ABB RobotStudio station: 4_28 - Copy_20220202-173113.rsstn

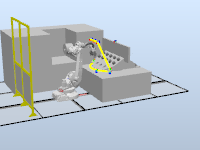
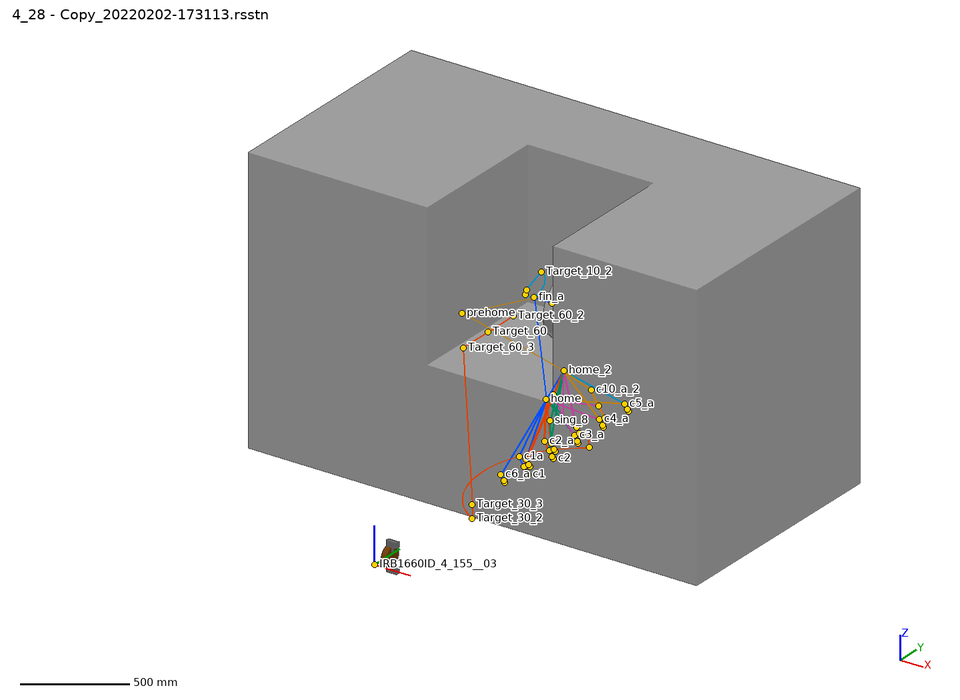
[picture v1: parts stored in the station drawn from their meshes, with robot base, taught points and paths (robot models come from the ABB library and are not in the file)]
Station Cambio_9_30 (saved by RobotStudio 21.4.9700.0)
Controller Controller3
  mechanical unit ROB_1: IRB1660ID_4_155__03, 6 joints, base frame (0, 0, 0) mm
Layout (positions relative to the parent item):
  - IRB1660ID_4_155__03 [mechanism, from Robots\IRB1660ID_4_155__03.rslib] at (0, 0, 0) mm; joint values [0.4367, 0.2271, -0.032, 0, 1.3757, 2.0075] (rad or m)
  - Pinza_1 [mechanism, from Efectores_finales - Copy\Pinza_1.rslib] at (900.75, 420.45, 1010) mm, rotated rx 180 ry 0 rz 90 deg; joint values [0, 0] (rad or m)
  - Conjunto_para_piezas_huecos [part] at (1981.81, -744.19, 0) mm, rotated rx 90 ry 0 rz 180 deg, size 1400 x 1300 x 1400 mm
  - Torno [part] at (-1172.42, 1966.27, 0) mm, rotated rx 0 ry 0 rz 180 deg, size 2500 x 1300 x 1500 mm
  - Fence_740 [graphiccomponentgroup, from Equipment\Fence_740.rslib] at (-1160.76, -802.49, 0) mm
    - Body 1 [part, from Equipment\Fence_740.rslib]
    - Body 2 [part, from Equipment\Fence_740.rslib]
  - Fence_2500 [graphiccomponentgroup, from Equipment\Fence_2500.rslib] at (1297.15, -826.85, 0) mm, rotated rx 0 ry 0 rz 90 deg
    - Body 1 [part, from Equipment\Fence_2500.rslib]
    - Body 2 [part, from Equipment\Fence_2500.rslib]
  - Fence_740_2 [graphiccomponentgroup, from Equipment\Fence_740.rslib] at (-1148.66, -57.63, 0) mm
    - Body 1 [part, from Equipment\Fence_740.rslib]
    - Body 2 [part, from Equipment\Fence_740.rslib]
  - c5 [part] at (1213.21, 355.81, 885.53) mm, rotated rx 0 ry -32 rz 0 deg, size 80 x 79.4 x 100 mm
  - c0 [part] at (367.03, 1016.09, 1000) mm, rotated rx -90 ry 0 rz 90 deg, size 80 x 79.4 x 100 mm
  - c8 [part] at (1084.59, -44.2, 808.36) mm, rotated rx 0 ry -32 rz 0 deg, size 80 x 79.4 x 100 mm
  - c4 [part] at (1213.21, 155.81, 885.53) mm, rotated rx 0 ry -32 rz 0 deg, size 80 x 79.4 x 100 mm
  - c7 [part] at (1084.59, -244.19, 808.36) mm, rotated rx 0 ry -32 rz 0 deg, size 80 x 79.4 x 100 mm
  - c6 [part] at (1084.59, -444.19, 808.36) mm, rotated rx 0 ry -32 rz 0 deg, size 80 x 79.4 x 100 mm
  - c9 [part] at (1084.59, 155.81, 808.36) mm, rotated rx 0 ry -32 rz 0 deg, size 80 x 79.4 x 100 mm
  - c10 [part] at (1084.59, 355.81, 808.36) mm, rotated rx 0 ry -32 rz 0 deg, size 80 x 79.4 x 100 mm
  - fin [part] at (377.58, 1016.27, 1000) mm, size 100 x 79.4 x 80 mm
  - c1 [part] at (1160.22, -444.2, 970.34) mm, rotated rx 90 ry 58 rz 0 deg, size 100 x 79.4 x 80 mm
  - Efector final 2 [part] at (70, 0, -80) mm, rotated rx 0 ry -90 rz -180 deg, size 100 x 99.5 x 30 mm
  - Pinza1_5 [part] at (130, 10, -10) mm, rotated rx 0 ry 0 rz 180 deg, size 60 x 20 x 60 mm
  - Pinza1_6 [part] at (130, -10, 150) mm, rotated rx 180 ry 0 rz 180 deg, size 60 x 20 x 60 mm
    - Pinza_2_1 [frame] at (30, 10, 80) mm, rotated rx 0 ry -90 rz 0 deg
  - Pinza_2 [mechanism, from Efectores_finales\PINZA2.rslib] at (900.75, 420.45, 1010) mm, rotated rx 180 ry 0 rz 90 deg; joint values [0, 0] (rad or m)
  - CollisionSensor [smart component, from Components\CollisionSensor.rslib]
      properties: Object1=Pinza_2; Object2=(none); NearMiss=0.0001; Part1=(none); Part2=(none); CollisionType=0
  - CollisionSensor_2 [smart component, from Components\CollisionSensor.rslib]
      properties: Object1=Pinza_2; Object2=c0_invisible; NearMiss=0.01; Part1=(none); Part2=(none); CollisionType=0
  - Attacher [smart component, from Components\Attacher.rslib]
      properties: Parent=Pinza_2; Flange=0; Child=(none); Mount=false; Offset=[0 0 0]; Orientation=[0 0 0]
  - Detacher [smart component, from Components\Detacher.rslib]
      properties: Child=(none); KeepPosition=true
  - CollisionSensor_3 [smart component, from Components\CollisionSensor.rslib]
      properties: Object1=Pinza_1; Object2=(none); NearMiss=0; Part1=(none); Part2=(none); CollisionType=0
  - Attacher_2 [smart component, from Components\Attacher.rslib]
      properties: Parent=Pinza_1; Flange=0; Child=(none); Mount=false; Offset=[0 0 0]; Orientation=[0 0 0]
  - Detacher_2 [smart component, from Components\Detacher.rslib]
      properties: Child=(none); KeepPosition=true
  - c2 [part] at (1207.14, -244.2, 895.25) mm, rotated rx 0 ry -32 rz 0 deg, size 80 x 79.4 x 100 mm
  - c0_invisible [part] at (277.58, 1016.27, 1000) mm, size 100 x 79.4 x 80 mm
  - CollisionSensor_4 [smart component, from Components\CollisionSensor.rslib]
      properties: Object1=Pinza_1; Object2=Conjunto_para_piezas_huecos; NearMiss=0.02; Part1=(none); Part2=(none); CollisionType=0
  - c3 [part] at (1213.21, -44.2, 885.53) mm, rotated rx 0 ry -32 rz 0 deg, size 80 x 79.4 x 100 mm
  - Hide [smart component, from Components\Hide.rslib]
      properties: Object=(none)
  - Show_2 [smart component, from Components\Show.rslib]
      properties: Object=Conjunto_para_piezas_huecos
  - visibilidad cilindros [smart component]
      signals: DI hide, DI show
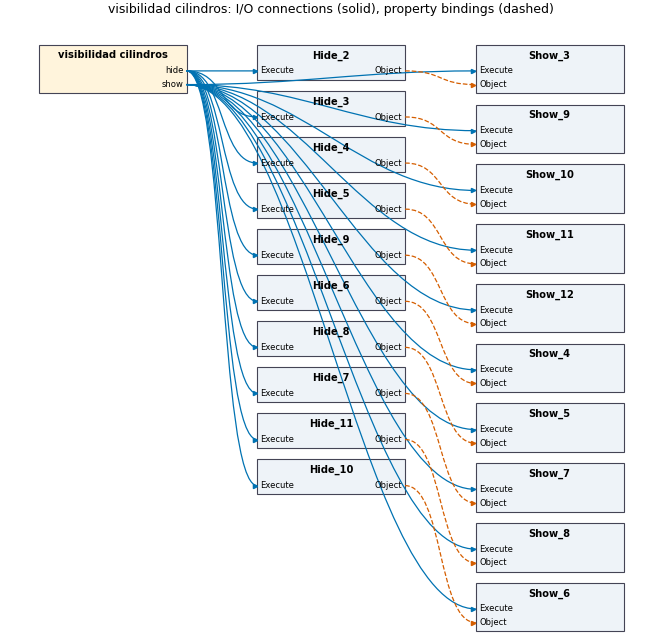
      connections:
        visibilidad cilindros.hide -> Hide_2.Execute
        visibilidad cilindros.hide -> Hide_3.Execute
        visibilidad cilindros.hide -> Hide_4.Execute
        visibilidad cilindros.hide -> Hide_5.Execute
        visibilidad cilindros.hide -> Hide_9.Execute
        visibilidad cilindros.hide -> Hide_6.Execute
        visibilidad cilindros.hide -> Hide_8.Execute
        visibilidad cilindros.hide -> Hide_7.Execute
        visibilidad cilindros.hide -> Hide_11.Execute
        visibilidad cilindros.show -> Show_3.Execute
        visibilidad cilindros.show -> Show_9.Execute
        visibilidad cilindros.show -> Show_10.Execute
        visibilidad cilindros.show -> Show_11.Execute
        visibilidad cilindros.show -> Show_12.Execute
        visibilidad cilindros.hide -> Hide_10.Execute
        visibilidad cilindros.show -> Show_4.Execute
        visibilidad cilindros.show -> Show_5.Execute
        visibilidad cilindros.show -> Show_6.Execute
        visibilidad cilindros.show -> Show_7.Execute
        visibilidad cilindros.show -> Show_8.Execute
        Hide_2.Object => Show_3.Object
        Hide_3.Object => Show_9.Object
        Hide_4.Object => Show_10.Object
        Hide_5.Object => Show_11.Object
        Hide_9.Object => Show_12.Object
        Hide_6.Object => Show_4.Object
        Hide_8.Object => Show_5.Object
        Hide_10.Object => Show_6.Object
        Hide_7.Object => Show_7.Object
        Hide_11.Object => Show_8.Object
    - Hide_2 [smart component, from Components\Hide.rslib]
        properties: Object=c1
    - Hide_3 [smart component, from Components\Hide.rslib]
        properties: Object=c2
    - Hide_4 [smart component, from Components\Hide.rslib]
        properties: Object=c3
    - Hide_5 [smart component, from Components\Hide.rslib]
        properties: Object=c4
    - Hide_6 [smart component, from Components\Hide.rslib]
        properties: Object=c6
    - Hide_7 [smart component, from Components\Hide.rslib]
        properties: Object=c9
    - Hide_8 [smart component, from Components\Hide.rslib]
        properties: Object=c7
    - Hide_9 [smart component, from Components\Hide.rslib]
        properties: Object=c5
    - Hide_10 [smart component, from Components\Hide.rslib]
        properties: Object=c8
    - Hide_11 [smart component, from Components\Hide.rslib]
        properties: Object=c10
    - Show_3 [smart component, from Components\Show.rslib]
        properties: Object=c1
    - Show_4 [smart component, from Components\Show.rslib]
        properties: Object=c6
    - Show_5 [smart component, from Components\Show.rslib]
        properties: Object=c7
    - Show_6 [smart component, from Components\Show.rslib]
        properties: Object=c8
    - Show_7 [smart component, from Components\Show.rslib]
        properties: Object=c9
    - Show_8 [smart component, from Components\Show.rslib]
        properties: Object=c10
    - Show_9 [smart component, from Components\Show.rslib]
        properties: Object=c2
    - Show_10 [smart component, from Components\Show.rslib]
        properties: Object=c3
    - Show_11 [smart component, from Components\Show.rslib]
        properties: Object=c4
    - Show_12 [smart component, from Components\Show.rslib]
        properties: Object=c5
  - mesa_giratoria_2 [smart component, from componentes\mesa_giratoria.rslib] at (1381.81, -44.2, 0) mm
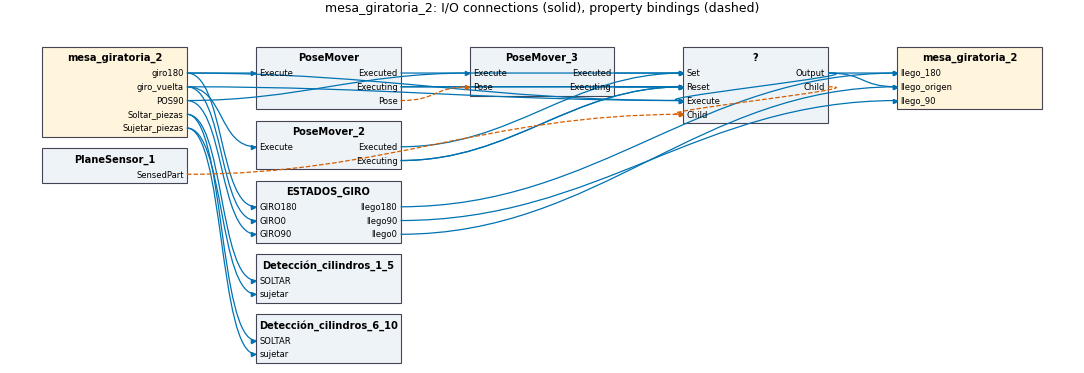
      connections:
        mesa_giratoria_2.giro180 -> PoseMover.Execute
        mesa_giratoria_2.giro_vuelta -> PoseMover_2.Execute
        PoseMover.Executed -> ?.Set
        ?.Output -> mesa_giratoria_2.llego_180
        PoseMover_2.Executed -> ?.Set
        ?.Output -> mesa_giratoria_2.llego_origen
        PoseMover_2.Executing -> ?.Reset
        PoseMover.Executing -> ?.Reset
        ?.Output -> ?.Execute
        mesa_giratoria_2.giro_vuelta -> ?.Execute
        mesa_giratoria_2.giro180 -> ?.Execute
        mesa_giratoria_2.POS90 -> PoseMover_3.Execute
        PoseMover_3.Executed -> ?.Set
        PoseMover.Executing -> ?.Reset
        PoseMover_2.Executing -> ?.Reset
        PoseMover_3.Executing -> ?.Reset
        PoseMover_3.Executing -> ?.Reset
        mesa_giratoria_2.giro180 -> ESTADOS_GIRO.GIRO180
        mesa_giratoria_2.giro_vuelta -> ESTADOS_GIRO.GIRO0
        mesa_giratoria_2.POS90 -> ESTADOS_GIRO.GIRO90
        ESTADOS_GIRO.llego180 -> mesa_giratoria_2.llego_180
        ESTADOS_GIRO.llego90 -> mesa_giratoria_2.llego_90
        ESTADOS_GIRO.llego0 -> mesa_giratoria_2.llego_origen
        mesa_giratoria_2.Soltar_piezas -> Detección_cilindros_1_5.SOLTAR
        mesa_giratoria_2.Soltar_piezas -> Detección_cilindros_6_10.SOLTAR
        mesa_giratoria_2.Sujetar_piezas -> Detección_cilindros_1_5.sujetar
        mesa_giratoria_2.Sujetar_piezas -> Detección_cilindros_6_10.sujetar
        PlaneSensor_1.SensedPart => ?.Child
        ?.Child => ?.Child
        PoseMover.Pose => PoseMover_3.Pose
    - Detección_cilindros_6_10 [smart component, from componentes\mesa_giratoria.rslib]
        connections:
          Detección_cilindros_6_10.SOLTAR -> Deteccion6.liberar
          Detección_cilindros_6_10.SOLTAR -> Deteccion10.liberar
          Detección_cilindros_6_10.SOLTAR -> Deteccion7.liberar
          Detección_cilindros_6_10.SOLTAR -> Deteccion8.liberar
          Detección_cilindros_6_10.SOLTAR -> Deteccion9.liberar
          Detección_cilindros_6_10.sujetar -> Deteccion6.Fijar
          Detección_cilindros_6_10.sujetar -> Deteccion10.Fijar
          Detección_cilindros_6_10.sujetar -> Deteccion7.Fijar
          Detección_cilindros_6_10.sujetar -> Deteccion9.Fijar
          Detección_cilindros_6_10.sujetar -> Deteccion8.Fijar
      - Deteccion6 [smart component, from componentes\mesa_giratoria.rslib]
        - Attacher_6 [smart component, from Components\Attacher.rslib]
            properties: Parent=Mi_mecanismo; Flange=0; Child=c6; Mount=false; Offset=[0 0 0]; Orientation=[0 0 0]
        - PlaneSensor_6 [smart component, from Components\PlaneSensor.rslib] at (-613.43, 800, 257.08) mm, rotated rx 0 ry 42 rz 0 deg
            properties: Origin=[0.0459897083517545 -0.4 1.14120505334971]; Axis1=[0.0787846202409767 0 0.0138918542133544]; Axis2=[0 0.04 0]; SensedPart=(none)
          - _sensorPart_ [part, from componentes\mesa_giratoria.rslib]
        - Detacher_6 [smart component, from Components\Detacher.rslib]
            properties: Child=(none); KeepPosition=true
      - Deteccion7 [smart component, from componentes\mesa_giratoria.rslib]
        - Attacher_7 [smart component, from Components\Attacher.rslib]
            properties: Parent=Mi_mecanismo; Flange=0; Child=c7; Mount=false; Offset=[0 0 0]; Orientation=[0 0 0]
        - PlaneSensor_7 [smart component, from Components\PlaneSensor.rslib] at (-613.43, 600, 257.08) mm, rotated rx 0 ry 42 rz 0 deg
            properties: Origin=[0.0459897083517545 -0.4 1.14120505334971]; Axis1=[0.0787846202409767 0 0.0138918542133544]; Axis2=[0 0.04 0]; SensedPart=(none)
          - _sensorPart_ [part, from componentes\mesa_giratoria.rslib]
        - Detacher_7 [smart component, from Components\Detacher.rslib]
            properties: Child=(none); KeepPosition=true
      - Deteccion8 [smart component, from componentes\mesa_giratoria.rslib]
        - Attacher_8 [smart component, from Components\Attacher.rslib]
            properties: Parent=Mi_mecanismo; Flange=0; Child=c8; Mount=false; Offset=[0 0 0]; Orientation=[0 0 0]
        - PlaneSensor_8 [smart component, from Components\PlaneSensor.rslib] at (-613.43, 400, 257.08) mm, rotated rx 0 ry 42 rz 0 deg
            properties: Origin=[0.0459897083517545 -0.4 1.14120505334971]; Axis1=[0.0787846202409767 0 0.0138918542133544]; Axis2=[0 0.04 0]; SensedPart=(none)
          - _sensorPart_ [part, from componentes\mesa_giratoria.rslib]
        - Detacher_8 [smart component, from Components\Detacher.rslib]
            properties: Child=(none); KeepPosition=true
      - Deteccion9 [smart component, from componentes\mesa_giratoria.rslib]
        - PlaneSensor_9 [smart component, from Components\PlaneSensor.rslib] at (-613.43, 0, 257.08) mm, rotated rx 0 ry 42 rz 0 deg
            properties: Origin=[0.0459897083517545 -0.4 1.14120505334971]; Axis1=[0.0787846202409767 0 0.0138918542133544]; Axis2=[0 0.04 0]; SensedPart=(none)
          - _sensorPart_ [part, from componentes\mesa_giratoria.rslib]
        - Attacher_9 [smart component, from Components\Attacher.rslib]
            properties: Parent=Mi_mecanismo; Flange=0; Child=c9; Mount=true; Offset=[0 0 0]; Orientation=[0 0 0]
        - Detacher_9 [smart component, from Components\Detacher.rslib]
            properties: Child=(none); KeepPosition=true
      - Deteccion10 [smart component, from componentes\mesa_giratoria.rslib]
        - Attacher_10 [smart component, from Components\Attacher.rslib] at (-100, -800, -200) mm
            properties: Parent=Mi_mecanismo; Flange=0; Child=c10; Mount=false; Offset=[0 0 0]; Orientation=[0 0 0]
        - PlaneSensor_10 [smart component, from Components\PlaneSensor.rslib] at (-613.43, 200, 257.08) mm, rotated rx 0 ry 42 rz 0 deg
            properties: Origin=[0.0459897083517545 -0.4 1.14120505334971]; Axis1=[0.0787846202409767 0 0.0138918542133544]; Axis2=[0 0.04 0]; SensedPart=(none)
          - _sensorPart_ [part, from componentes\mesa_giratoria.rslib]
        - Detacher_10 [smart component, from Components\Detacher.rslib]
            properties: Child=(none); KeepPosition=true
    - Detección_cilindros_1_5 [smart component, from componentes\mesa_giratoria.rslib]
        connections:
          PlaneSensor_1.SensorOut -> Attacher_1.Execute
          PlaneSensor_2.SensorOut -> Attacher_2.Execute
          PlaneSensor_3.SensorOut -> Attacher_3.Execute
          PlaneSensor_4.SensorOut -> Attacher_4.Execute
          PlaneSensor_5.SensorOut -> Attacher_5.Execute
          Detección_cilindros_1_5.SOLTAR -> Deteccion1.liberar
          Detección_cilindros_1_5.sujetar -> Deteccion1.Fijar
          Detección_cilindros_1_5.SOLTAR -> Deteccion2.liberar
          Detección_cilindros_1_5.sujetar -> Deteccion2.Fijar
          Detección_cilindros_1_5.SOLTAR -> Deteccion3.liberar
          Detección_cilindros_1_5.sujetar -> Deteccion3.Fijar
          Detección_cilindros_1_5.SOLTAR -> Deteccion4.liberar
          Detección_cilindros_1_5.sujetar -> Deteccion4.Fijar
          Detección_cilindros_1_5.SOLTAR -> Deteccion5.liberar
          Detección_cilindros_1_5.sujetar -> Deteccion5.Fijar
          Attacher_1.Parent => Attacher_2.Parent
          Attacher_2.Parent => Attacher_3.Parent
          Attacher_3.Parent => Attacher_4.Parent
          Attacher_4.Parent => Attacher_5.Parent
      - Deteccion1 [smart component, from componentes\mesa_giratoria.rslib]
          connections:
            Deteccion1.liberar -> Detacher_1.Execute
            Deteccion1.Fijar -> Attacher_2.Execute
            Attacher_1.Child => Detacher_1.Child
            PlaneSensor_1.SensedPart => Attacher_2.Child
        - Attacher_1 [smart component, from Components\Attacher.rslib] at (-100, 0, -200) mm
            properties: Parent=Mi_mecanismo; Flange=0; Child=c1; Mount=false; Offset=[0 0 0]; Orientation=[0 0 0]
        - PlaneSensor_1 [smart component, from Components\PlaneSensor.rslib] at (-742.06, 0, 334.25) mm, rotated rx 0 ry 42 rz 0 deg
            properties: Origin=[0.0459897083517545 -0.4 1.14120505334971]; Axis1=[0.0787846202409767 0 0.0138918542133544]; Axis2=[0 0.04 0]; SensedPart=(none)
          - _sensorPart_ [part, from componentes\mesa_giratoria.rslib]
        - Detacher_1 [smart component, from Components\Detacher.rslib]
            properties: Child=c1; KeepPosition=true
        - Attacher_2 [smart component, from Components\Attacher.rslib]
            properties: Parent=(none); Flange=0; Child=(none); Mount=false; Offset=[0 0 0]; Orientation=[0 0 0]
      - Deteccion2 [smart component, from componentes\mesa_giratoria.rslib]
          connections:
            Deteccion2.liberar -> Detacher_2.Execute
            Attacher_2.Child => Detacher_2.Child
        - Attacher_2 [smart component, from Components\Attacher.rslib] at (-100, 0, -200) mm
            properties: Parent=Mi_mecanismo; Flange=0; Child=c2; Mount=false; Offset=[0 0 0]; Orientation=[0 0 0]
        - PlaneSensor_2 [smart component, from Components\PlaneSensor.rslib] at (-742.06, 200, 334.25) mm, rotated rx 0 ry 42 rz 0 deg
            properties: Origin=[0.0459897083517545 -0.4 1.14120505334971]; Axis1=[0.0787846202409767 0 0.0138918542133544]; Axis2=[0 0.04 0]; SensedPart=(none)
          - _sensorPart_ [part, from componentes\mesa_giratoria.rslib]
        - Detacher_2 [smart component, from Components\Detacher.rslib]
            properties: Child=c2; KeepPosition=true
      - Deteccion3 [smart component, from componentes\mesa_giratoria.rslib]
        - Attacher_3 [smart component, from Components\Attacher.rslib]
            properties: Parent=Mi_mecanismo; Flange=0; Child=c3; Mount=false; Offset=[0 0 0]; Orientation=[0 0 0]
        - PlaneSensor_3 [smart component, from Components\PlaneSensor.rslib] at (-742.06, 400, 334.25) mm, rotated rx 0 ry 42 rz 0 deg
            properties: Origin=[0.0459897083517545 -0.4 1.14120505334971]; Axis1=[0.0787846202409767 0 0.0138918542133544]; Axis2=[0 0.04 0]; SensedPart=(none)
          - _sensorPart_ [part, from componentes\mesa_giratoria.rslib]
        - Detacher_3 [smart component, from Components\Detacher.rslib]
            properties: Child=(none); KeepPosition=true
      - Deteccion4 [smart component, from componentes\mesa_giratoria.rslib]
        - Attacher_4 [smart component, from Components\Attacher.rslib]
            properties: Parent=Mi_mecanismo; Flange=0; Child=c4; Mount=false; Offset=[0 0 0]; Orientation=[0 0 0]
        - PlaneSensor_4 [smart component, from Components\PlaneSensor.rslib] at (-742.06, 600, 334.25) mm, rotated rx 0 ry 42 rz 0 deg
            properties: Origin=[0.0459897083517545 -0.4 1.14120505334971]; Axis1=[0.0787846202409767 0 0.0138918542133544]; Axis2=[0 0.04 0]; SensedPart=(none)
          - _sensorPart_ [part, from componentes\mesa_giratoria.rslib]
        - Detacher_4 [smart component, from Components\Detacher.rslib]
            properties: Child=(none); KeepPosition=true
      - Deteccion5 [smart component, from componentes\mesa_giratoria.rslib]
        - Attacher_5 [smart component, from Components\Attacher.rslib]
            properties: Parent=Mi_mecanismo; Flange=0; Child=c5; Mount=false; Offset=[0 0 0]; Orientation=[0 0 0]
        - PlaneSensor_5 [smart component, from Components\PlaneSensor.rslib] at (-742.06, 800, 334.25) mm, rotated rx 0 ry 42 rz 0 deg
            properties: Origin=[0.0459897083517545 -0.4 1.14120505334971]; Axis1=[0.0787846202409767 0 0.0138918542133544]; Axis2=[0 0.04 0]; SensedPart=(none)
          - _sensorPart_ [part, from componentes\mesa_giratoria.rslib]
        - Detacher_5 [smart component, from Components\Detacher.rslib]
            properties: Child=(none); KeepPosition=true
    - Mi_mecanismo [mechanism, from componentes\mesa_giratoria.rslib] at (-100, 0, -200) mm; joint values [0, 0] (rad or m)
    - ESTADOS_GIRO [smart component, from componentes\mesa_giratoria.rslib]
        connections:
          ESTADOS_GIRO.GIRO180 -> PoseMover.Execute
          ESTADOS_GIRO.GIRO90 -> PoseMover_3.Execute
          ESTADOS_GIRO.GIRO0 -> PoseMover_2.Execute
          PoseMover.Executing -> LogicSRLatch_6.Reset
          PoseMover.Executing -> LogicSRLatch_4.Reset
          PoseMover.Executed -> LogicSRLatch_5.Set
          PoseMover_3.Executed -> LogicSRLatch_6.Set
          PoseMover_2.Executed -> LogicSRLatch_4.Set
          PoseMover_3.Executing -> LogicSRLatch_5.Reset
          PoseMover_3.Executing -> LogicSRLatch_4.Reset
          PoseMover_2.Executing -> LogicSRLatch_6.Reset
          PoseMover_2.Executing -> LogicSRLatch_5.Reset
          LogicSRLatch_5.Output -> ESTADOS_GIRO.llego180
          LogicSRLatch_6.Output -> ESTADOS_GIRO.llego90
          LogicSRLatch_4.Output -> ESTADOS_GIRO.llego0
      - PoseMover [smart component, from Components\PoseMover.rslib]
          properties: Mechanism=Mi_mecanismo; Pose=1; Duration=4
      - PoseMover_2 [smart component, from Components\PoseMover.rslib]
          properties: Mechanism=Mi_mecanismo; Pose=2; Duration=4
      - PoseMover_3 [smart component, from Components\PoseMover.rslib]
          properties: Mechanism=Mi_mecanismo; Pose=3; Duration=4
      - LogicSRLatch_4 [smart component, from Components\LogicSRLatch.rslib]
      - LogicSRLatch_5 [smart component, from Components\LogicSRLatch.rslib]
      - LogicSRLatch_6 [smart component, from Components\LogicSRLatch.rslib]
    - c10_1 [part, from componentes\mesa_giratoria.rslib] at (197.22, -400, 1008.36) mm, rotated rx 0 ry -30 rz 180 deg
    - c10 [part, from componentes\mesa_giratoria.rslib] at (-297.22, 400, 808.36) mm, rotated rx 0 ry -30 rz 0 deg
    - c9_1 [part, from componentes\mesa_giratoria.rslib] at (197.22, -200, 1008.36) mm, rotated rx 0 ry 30 rz 0 deg
    - c9 [part, from componentes\mesa_giratoria.rslib] at (-297.22, 200, 808.36) mm, rotated rx 0 ry 30 rz 180 deg
    - c8_1 [part, from componentes\mesa_giratoria.rslib] at (197.95, 0, 1007.93) mm, rotated rx 0 ry 30 rz 0 deg
    - c8 [part, from componentes\mesa_giratoria.rslib] at (-297.95, 0, 807.93) mm, rotated rx 0 ry 30 rz 180 deg
    - c7_1 [part, from componentes\mesa_giratoria.rslib] at (197.22, 200, 1008.36) mm, rotated rx 0 ry -30 rz 180 deg
    - c7 [part, from componentes\mesa_giratoria.rslib] at (-297.22, -200, 808.36) mm, rotated rx 0 ry -30 rz 0 deg
    - c6_1 [part, from componentes\mesa_giratoria.rslib] at (197.22, 400, 1008.36) mm, rotated rx 0 ry -30 rz 180 deg
    - c6 [part, from componentes\mesa_giratoria.rslib] at (-297.22, -400, 808.36) mm, rotated rx 0 ry -30 rz 0 deg
    - c5_1 [part, from componentes\mesa_giratoria.rslib] at (68.6, 400, 1085.53) mm, rotated rx 0 ry -30 rz 180 deg
    - c5 [part, from componentes\mesa_giratoria.rslib] at (-168.6, -400, 885.53) mm, rotated rx 0 ry -30 rz 0 deg
    - c4_1 [part, from componentes\mesa_giratoria.rslib] at (68.6, 200, 1085.53) mm, rotated rx 0 ry -30 rz 180 deg
    - c4 [part, from componentes\mesa_giratoria.rslib] at (-168.6, -200, 885.53) mm, rotated rx 0 ry -30 rz 0 deg
    - c3_1 [part, from componentes\mesa_giratoria.rslib] at (-31.4, 0, 885.53) mm, rotated rx 0 ry -30 rz 180 deg
    - c3 [part, from componentes\mesa_giratoria.rslib] at (-168.6, 0, 885.53) mm, rotated rx 0 ry -30 rz 0 deg
    - c2_1 [part, from componentes\mesa_giratoria.rslib] at (-31.4, -200, 885.53) mm, rotated rx 0 ry -30 rz 180 deg
    - c2 [part, from componentes\mesa_giratoria.rslib] at (-168.6, 200, 885.53) mm, rotated rx 0 ry -30 rz 0 deg
    - c1_1 [part, from componentes\mesa_giratoria.rslib] at (-31.4, -400, 885.53) mm, rotated rx 0 ry -30 rz 180 deg
    - c1 [part, from componentes\mesa_giratoria.rslib] at (-168.6, 400, 885.53) mm, rotated rx 0 ry -30 rz 0 deg
Attachment: Pinza_2 is attached to IRB1660ID_4_155__03 / Link6
Attachment: Pinza_1 is attached to IRB1660ID_4_155__03 / Link6
Attachment: Attacher_10 is attached to c6
Attachment: Attacher_1 is attached to Mi_mecanismo / L3
Attachment: Attacher_2 is attached to Mi_mecanismo / L3
Attachment: c10 is attached to Mi_mecanismo / L3
Attachment: c9 is attached to Mi_mecanismo / L3
Attachment: c8 is attached to Mi_mecanismo / L3
Attachment: c7 is attached to Mi_mecanismo / L3
Attachment: c6 is attached to Mi_mecanismo / L3
Attachment: c5 is attached to Mi_mecanismo / L3
Attachment: c4 is attached to Mi_mecanismo / L3
Attachment: c3 is attached to Mi_mecanismo / L3
Attachment: c2 is attached to Mi_mecanismo / L3
Attachment: c1 is attached to Mi_mecanismo / L3
Attachment: mesa_giratoria_2 is attached to c7_1
Station signals: DO s, DI signal
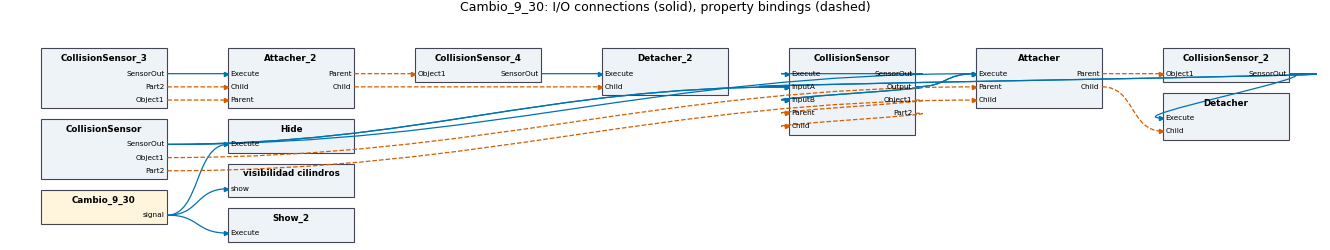
Station logic (signal -> signal, property => property):
  CollisionSensor.SensorOut -> Attacher.Execute
  CollisionSensor_3.SensorOut -> Attacher_2.Execute
  LogicGate_2.Output -> Attacher.Execute
  CollisionSensor_2.SensorOut -> LogicGate.InputA
  LogicGate.Output -> LogicGate_2.InputB
  CollisionSensor.SensorOut -> LogicGate_2.InputA
  CollisionSensor.SensorOut -> LogicGate_4.InputA
  CollisionSensor_2.SensorOut -> LogicGate_3.InputA
  LogicGate_3.Output -> LogicGate_4.InputB
  LogicGate_4.Output -> Attacher.Execute
  CollisionSensor_2.SensorOut -> Detacher.Execute
  CollisionSensor.SensorOut -> Attacher.Execute
  CollisionSensor_4.SensorOut -> Detacher_2.Execute
  Cambio_9_30.signal -> Hide.Execute
  Cambio_9_30.signal -> visibilidad cilindros.show
  Cambio_9_30.signal -> Show_2.Execute
  CollisionSensor.Object1 => Attacher.Parent
  CollisionSensor.Part2 => Attacher.Child
  CollisionSensor.Object1 => Attacher.Parent
  CollisionSensor.Part2 => Attacher.Child
  CollisionSensor_3.Part2 => Attacher_2.Child
  CollisionSensor_3.Object1 => Attacher_2.Parent
  Attacher.Parent => CollisionSensor_2.Object1
  Attacher.Child => Detacher.Child
  Attacher_2.Parent => CollisionSensor_4.Object1
  Attacher_2.Child => Detacher_2.Child
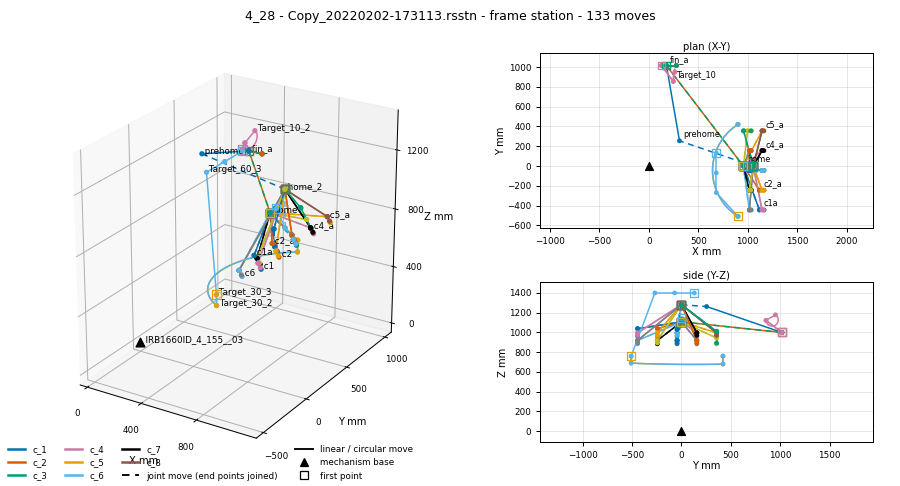
[picture p0: tool path of 4_28 - Copy_20220202-173113.rsstn in frame station, 133 of 133 moves have a stored position in this frame; points joined in program order, loops and branches not executed]
Targets, tools, work objects and paths stored in the station, written as RAPID:
! task T_ROB1
MODULE Module1
  CONST robtarget home:=[[955.495207776,0,1107.397459622],[0.258819045,0,-0.965925826,0],[0,0,0,0],[9E+09,9E+09,9E+09,9E+09,9E+09,9E+09]];
  CONST robtarget c1:=[[1165.520192645,-444.195,961.85451904],[0.275637356,0,0.961261696,0],[-1,1,-2,0],[9E+09,9E+09,9E+09,9E+09,9E+09,9E+09]];
  CONST robtarget c1a:=[[1117.82745884,-444.195,1038.178847679],[0.275637356,0,0.961261696,0],[-1,1,-2,0],[9E+09,9E+09,9E+09,9E+09,9E+09,9E+09]];
  CONST robtarget c2:=[[1165.520192645,-244.195,961.85451904],[0.275637356,0,0.961261696,0],[-1,1,-2,0],[9E+09,9E+09,9E+09,9E+09,9E+09,9E+09]];
  CONST robtarget c2_a:=[[1117.82745884,-244.195,1038.178847679],[0.275637356,0,0.961261696,0],[-1,1,-2,0],[9E+09,9E+09,9E+09,9E+09,9E+09,9E+09]];
  CONST robtarget c3:=[[1165.520192645,-44.195,961.85451904],[0.275637356,0,0.961261696,0],[-1,-1,0,1],[9E+09,9E+09,9E+09,9E+09,9E+09,9E+09]];
  CONST robtarget c3_a:=[[1144.323422065,-44.195,995.776442879],[0.275637356,0,0.961261696,0],[-1,-1,0,1],[9E+09,9E+09,9E+09,9E+09,9E+09,9E+09]];
  CONST robtarget c4:=[[1165.520192645,155.805,961.85451904],[0.275637356,0,0.961261696,0],[0,-2,1,0],[9E+09,9E+09,9E+09,9E+09,9E+09,9E+09]];
  CONST robtarget c4_a:=[[1144.323422065,155.805,995.776442879],[0.275637356,0,0.961261696,0],[0,-2,1,0],[9E+09,9E+09,9E+09,9E+09,9E+09,9E+09]];
  CONST robtarget c5:=[[1165.520192645,355.805,961.85451904],[0.275637356,0,0.961261696,0],[0,-2,1,0],[9E+09,9E+09,9E+09,9E+09,9E+09,9E+09]];
  CONST robtarget c5_a:=[[1144.323422065,355.805,995.77644288],[0.275637356,0,0.961261696,0],[0,-2,1,0],[9E+09,9E+09,9E+09,9E+09,9E+09,9E+09]];
  CONST robtarget c6:=[[1036.896192645,-444.195,884.68051904],[0.275637356,0,0.961261696,0],[-1,1,-2,0],[9E+09,9E+09,9E+09,9E+09,9E+09,9E+09]];
  CONST robtarget c6_a:=[[1015.699422065,-444.195,918.60244288],[0.275637356,0,0.961261696,0],[-1,1,-2,0],[9E+09,9E+09,9E+09,9E+09,9E+09,9E+09]];
  CONST robtarget c7:=[[1036.896192645,-244.195,884.68051904],[0.275637356,0,0.961261696,0],[-1,1,-2,0],[9E+09,9E+09,9E+09,9E+09,9E+09,9E+09]];
  CONST robtarget c7_a:=[[1015.699422065,-244.195,918.60244288],[0.275637356,0,0.961261696,0],[-1,1,-2,0],[9E+09,9E+09,9E+09,9E+09,9E+09,9E+09]];
  CONST robtarget c8:=[[1036.896192645,-44.195,884.68051904],[0.275637356,0,0.961261696,0],[-1,-1,0,1],[9E+09,9E+09,9E+09,9E+09,9E+09,9E+09]];
  CONST robtarget c8_a:=[[1015.699422065,-44.195,918.60244288],[0.275637356,0,0.961261696,0],[-1,-1,0,1],[9E+09,9E+09,9E+09,9E+09,9E+09,9E+09]];
  CONST robtarget c9_a:=[[1015.699422065,155.805,918.60244288],[0.275637356,0,0.961261696,0],[0,-2,1,0],[9E+09,9E+09,9E+09,9E+09,9E+09,9E+09]];
  CONST robtarget c9:=[[1036.896192645,155.805,884.68051904],[0.275637356,0,0.961261696,0],[0,-2,1,0],[9E+09,9E+09,9E+09,9E+09,9E+09,9E+09]];
  CONST robtarget c10:=[[1036.896192645,355.805,884.68051904],[0.275637356,0,0.961261696,0],[0,-2,1,0],[9E+09,9E+09,9E+09,9E+09,9E+09,9E+09]];
  CONST robtarget c10_a:=[[999.80184413,355.805,944.043885759],[0.275637356,0,0.961261696,0],[0,-2,1,0],[9E+09,9E+09,9E+09,9E+09,9E+09,9E+09]];
  CONST robtarget fin_a:=[[177.584,1016.268,1000],[0.5,0.5,0.5,0.5],[0,1,-1,0],[9E+09,9E+09,9E+09,9E+09,9E+09,9E+09]];
  CONST robtarget fin:=[[277.584,1016.268,1000],[0.5,0.5,0.5,0.5],[0,1,-1,0],[9E+09,9E+09,9E+09,9E+09,9E+09,9E+09]];
  CONST robtarget home_2:=[[1055.495207776,0,1280.602540378],[0.965925826,0,0.258819045,0],[0,0,0,0],[9E+09,9E+09,9E+09,9E+09,9E+09,9E+09]];
  CONST robtarget final_a:=[[177.584,1016.268,1000],[0.5,-0.5,0.5,-0.5],[0,0,0,0],[9E+09,9E+09,9E+09,9E+09,9E+09,9E+09]];
  CONST robtarget final:=[[278.084,1016.268,1000],[0.5,-0.5,0.5,-0.5],[0,1,1,0],[9E+09,9E+09,9E+09,9E+09,9E+09,9E+09]];
  CONST robtarget prehome:=[[309.604,254.998,1262.538],[0.396697298,0.585347123,0.410036045,0.576081975],[0,1,0,0],[9E+09,9E+09,9E+09,9E+09,9E+09,9E+09]];
  CONST robtarget c1_3:=[[1160.221,-444.195,970.335],[0,0.961261696,0,0.275637356],[-1,1,0,0],[9E+09,9E+09,9E+09,9E+09,9E+09,9E+09]];
  CONST robtarget c1a_3:=[[1144.323422065,-444.195,995.77644288],[0,0.961261696,0,0.275637356],[-1,1,0,0],[9E+09,9E+09,9E+09,9E+09,9E+09,9E+09]];
  CONST robtarget c2_3:=[[1160.221,-244.195,970.335],[0,0.961261696,0,0.275637356],[-1,1,0,0],[9E+09,9E+09,9E+09,9E+09,9E+09,9E+09]];
  CONST robtarget c2_a_2:=[[1144.323422065,-244.195,995.77644288],[0,0.961261696,0,0.275637356],[-1,1,0,0],[9E+09,9E+09,9E+09,9E+09,9E+09,9E+09]];
  CONST robtarget c3_3:=[[1160.221,-44.195,970.335],[0,0.961261696,0,0.275637356],[-1,-1,-2,1],[9E+09,9E+09,9E+09,9E+09,9E+09,9E+09]];
  CONST robtarget c3_a_2:=[[1144.323422065,-44.195,995.77644288],[0,0.961261696,0,0.275637356],[-1,-1,-2,1],[9E+09,9E+09,9E+09,9E+09,9E+09,9E+09]];
  CONST robtarget c4_3:=[[1160.221,155.805,970.335],[0,0.961261696,0,0.275637356],[0,-2,-1,0],[9E+09,9E+09,9E+09,9E+09,9E+09,9E+09]];
  CONST robtarget c4_a_2:=[[1144.323422065,155.805,995.77644288],[0,0.961261696,0,0.275637356],[0,-2,-1,0],[9E+09,9E+09,9E+09,9E+09,9E+09,9E+09]];
  CONST robtarget c5_3:=[[1160.221,355.805,970.335],[0,0.961261696,0,0.275637356],[0,-2,-1,0],[9E+09,9E+09,9E+09,9E+09,9E+09,9E+09]];
  CONST robtarget c5_a_2:=[[1144.323422065,355.805,995.77644288],[0,0.961261696,0,0.275637356],[0,-2,-1,0],[9E+09,9E+09,9E+09,9E+09,9E+09,9E+09]];
  CONST robtarget c6_3:=[[1031.597,-444.195,893.161],[0,0.961261696,0,0.275637356],[-1,1,0,0],[9E+09,9E+09,9E+09,9E+09,9E+09,9E+09]];
  CONST robtarget c6_a_2:=[[1015.699422065,-444.195,918.60244288],[0,0.961261696,0,0.275637356],[-1,1,0,0],[9E+09,9E+09,9E+09,9E+09,9E+09,9E+09]];
  CONST robtarget c7_3:=[[1031.597,-244.195,893.161],[0,0.961261696,0,0.275637356],[-1,1,0,0],[9E+09,9E+09,9E+09,9E+09,9E+09,9E+09]];
  CONST robtarget c7_a_2:=[[1015.699422065,-244.195,918.60244288],[0,0.961261696,0,0.275637356],[-1,1,0,0],[9E+09,9E+09,9E+09,9E+09,9E+09,9E+09]];
  CONST robtarget c8_3:=[[1031.597,-44.195,893.161],[0,0.961261696,0,0.275637356],[-1,-1,-2,1],[9E+09,9E+09,9E+09,9E+09,9E+09,9E+09]];
  CONST robtarget c8_a_2:=[[1015.699422065,-44.195,918.60244288],[0,0.961261696,0,0.275637356],[-1,-1,-2,1],[9E+09,9E+09,9E+09,9E+09,9E+09,9E+09]];
  CONST robtarget c9_2:=[[1031.597,155.805,893.161],[0,0.961261696,0,0.275637356],[0,-2,-1,0],[9E+09,9E+09,9E+09,9E+09,9E+09,9E+09]];
  CONST robtarget c9_a_3:=[[1015.699422065,155.805,918.60244288],[0,0.961261696,0,0.275637356],[0,-2,-1,0],[9E+09,9E+09,9E+09,9E+09,9E+09,9E+09]];
  CONST robtarget c10_3:=[[1031.597,355.805,893.161],[0,0.961261696,0,0.275637356],[0,-2,-1,0],[9E+09,9E+09,9E+09,9E+09,9E+09,9E+09]];
  CONST robtarget c10_a_2:=[[957.40830297,355.805,1011.88773344],[0,0.961261696,0,0.275637356],[0,-2,-1,0],[9E+09,9E+09,9E+09,9E+09,9E+09,9E+09]];
  CONST robtarget singular:=[[794.078577227,72.053971449,1440.197967774],[0.008993924,0.229595419,-0.191275883,-0.954263375],[-1,-1,1,1],[9E+09,9E+09,9E+09,9E+09,9E+09,9E+09]];
  CONST robtarget sing:=[[996.034157953,0.89711627,1142.308388844],[0.004439032,-0.989602616,0.000644854,0.143758623],[0,-1,-2,0],[9E+09,9E+09,9E+09,9E+09,9E+09,9E+09]];
  CONST robtarget c3_a_2_2:=[[1086.031473643,-43.527299213,1055.048962422],[0.000858943,0.974553856,-0.004750994,0.224101477],[-1,-1,-2,1],[9E+09,9E+09,9E+09,9E+09,9E+09,9E+09]];
  CONST robtarget sing_8:=[[1009.414631395,-44.524440453,1031.444612597],[0.010580344,0.969216357,0.000547425,0.245982539],[-1,-1,-2,1],[9E+09,9E+09,9E+09,9E+09,9E+09,9E+09]];
  CONST robtarget Target_10:=[[246.795972221,856.078436824,1122.33728984],[0.491799027,0.566655461,0.470411016,0.464487654],[0,1,-2,0],[9E+09,9E+09,9E+09,9E+09,9E+09,9E+09]];
  CONST robtarget Target_10_2:=[[263.201550694,951.392827128,1178.426718398],[0.491799027,0.566655461,0.470411016,0.464487654],[0,1,-2,0],[9E+09,9E+09,9E+09,9E+09,9E+09,9E+09]];
  CONST robtarget Target_10_3:=[[255.576271719,958.762265661,1078.990575592],[0.491799027,0.566655461,0.470411016,0.464487654],[0,1,-2,0],[9E+09,9E+09,9E+09,9E+09,9E+09,9E+09]];
  CONST robtarget Target_20:=[[127.584052063,1016.268015631,999.999997056],[0.499999999,0.500000042,0.500000004,0.499999956],[0,1,-2,0],[9E+09,9E+09,9E+09,9E+09,9E+09,9E+09]];
  CONST robtarget Target_30:=[[900.746,-508.84,720],[0,1,0,0],[0,0,0,0],[9E+09,9E+09,9E+09,9E+09,9E+09,9E+09]];
  CONST robtarget Target_40:=[[900.746,420.45,720],[0,1,0,0],[0,0,1,0],[9E+09,9E+09,9E+09,9E+09,9E+09,9E+09]];
  CONST robtarget Target_50:=[[675.669,-229.408,680],[0,1,0,0],[-1,0,0,0],[9E+09,9E+09,9E+09,9E+09,9E+09,9E+09]];
  CONST robtarget Target_30_2:=[[900.746,-508.84,690],[0,1,0,0],[-1,0,0,0],[9E+09,9E+09,9E+09,9E+09,9E+09,9E+09]];
  CONST robtarget Target_40_2:=[[900.746,420.45,680],[0,1,0,0],[0,0,1,0],[9E+09,9E+09,9E+09,9E+09,9E+09,9E+09]];
  CONST robtarget Target_30_3:=[[900.746,-508.84,760],[0,1,0,0],[-1,0,0,0],[9E+09,9E+09,9E+09,9E+09,9E+09,9E+09]];
  CONST robtarget Target_40_3:=[[900.746,420.45,760],[0,1,0,0],[0,0,1,0],[9E+09,9E+09,9E+09,9E+09,9E+09,9E+09]];
  CONST robtarget Target_60:=[[681.812,-69.195,1400],[0.707106781,0,0.707106781,0],[-1,0,-2,0],[9E+09,9E+09,9E+09,9E+09,9E+09,9E+09]];
  CONST robtarget Target_60_2:=[[681.812,130.805,1400],[0.707106781,0,0.707106781,0],[0,-1,-1,0],[9E+09,9E+09,9E+09,9E+09,9E+09,9E+09]];
  CONST robtarget Target_60_3:=[[681.812,-269.195,1400],[0.707106781,0,0.707106781,0],[-1,0,-2,0],[9E+09,9E+09,9E+09,9E+09,9E+09,9E+09]];
  PROC c_1()
    MoveJ home,v1000,z100,Pinza_2_1\WObj:=Workobject_2;
    MoveL c1a,v1000,z100,Pinza_2_1\WObj:=Workobject_2;
    MoveL c1,v1000,fine,Pinza_2_1\WObj:=Workobject_2;
    MoveL c1a,v1000,z100,Pinza_2_1\WObj:=Workobject_2;
    MoveJ home,v1000,z100,Pinza_2_1\WObj:=Workobject_2;
  ENDPROC
  PROC c_2()
    MoveJ home,v1000,z100,Pinza_2_1\WObj:=Workobject_2;
    MoveL c2_a,v1000,z100,Pinza_2_1\WObj:=Workobject_2;
    MoveL c2,v1000,z100,Pinza_2_1\WObj:=Workobject_2;
    MoveL c2_a,v1000,z100,Pinza_2_1\WObj:=Workobject_2;
    MoveJ home,v1000,z100,Pinza_2_1\WObj:=Workobject_2;
  ENDPROC
  PROC c_3()
    MoveJ home,v1000,z100,Pinza_2_1\WObj:=Workobject_2;
    MoveJ c3_a,v1000,z100,Pinza_2_1\WObj:=Workobject_2;
    MoveL c3,v1000,z100,Pinza_2_1\WObj:=Workobject_2;
    MoveJ c3_a,v1000,z100,Pinza_2_1\WObj:=Workobject_2;
    MoveJ home,v1000,z100,Pinza_2_1\WObj:=Workobject_2;
  ENDPROC
  PROC c_4()
    MoveJ home,v1000,z100,Pinza_2_1\WObj:=Workobject_2;
    MoveL c4_a,v1000,z100,Pinza_2_1\WObj:=Workobject_2;
    MoveL c4,v1000,z100,Pinza_2_1\WObj:=Workobject_2;
    MoveL c4_a,v1000,z100,Pinza_2_1\WObj:=Workobject_2;
    MoveJ home,v1000,z100,Pinza_2_1\WObj:=Workobject_2;
  ENDPROC
  PROC c_5()
    MoveJ home,v1000,z100,Pinza_2_1\WObj:=Workobject_2;
    MoveL c5_a,v1000,z100,Pinza_2_1\WObj:=Workobject_2;
    MoveL c5,v1000,z100,Pinza_2_1\WObj:=Workobject_2;
    MoveL c5_a,v1000,z100,Pinza_2_1\WObj:=Workobject_2;
    MoveJ home,v1000,z100,Pinza_2_1\WObj:=Workobject_2;
  ENDPROC
  PROC c_6()
    MoveJ home,v1000,z100,Pinza_2_1\WObj:=Workobject_2;
    MoveL c6_a,v1000,z100,Pinza_2_1\WObj:=Workobject_2;
    MoveL c6,v1000,z100,Pinza_2_1\WObj:=Workobject_2;
    MoveL c6_a,v1000,z100,Pinza_2_1\WObj:=Workobject_2;
    MoveJ home,v1000,z100,Pinza_2_1\WObj:=Workobject_2;
  ENDPROC
  PROC c_7()
    MoveJ home,v1000,z100,Pinza_2_1\WObj:=Workobject_2;
    MoveL c7_a,v1000,z100,Pinza_2_1\WObj:=Workobject_2;
    MoveL c7,v1000,z100,Pinza_2_1\WObj:=Workobject_2;
    MoveL c7_a,v1000,z100,Pinza_2_1\WObj:=Workobject_2;
    MoveJ home,v1000,z100,Pinza_2_1\WObj:=Workobject_2;
  ENDPROC
  PROC c_8()
    MoveJ home,v1000,z100,Pinza_2_1\WObj:=Workobject_2;
    MoveJ c8_a,v1000,z100,Pinza_2_1\WObj:=Workobject_2;
    MoveL c8,v1000,z100,Pinza_2_1\WObj:=Workobject_2;
    MoveJ c8_a,v1000,z100,Pinza_2_1\WObj:=Workobject_2;
    MoveJ home,v1000,z100,Pinza_2_1\WObj:=Workobject_2;
  ENDPROC
  PROC c_9()
    MoveJ home,v1000,z100,Pinza_2_1\WObj:=Workobject_2;
    MoveL c9_a,v1000,z100,Pinza_2_1\WObj:=Workobject_2;
    MoveL c9,v1000,z100,Pinza_2_1\WObj:=Workobject_2;
    MoveL c9_a,v1000,z100,Pinza_2_1\WObj:=Workobject_2;
    MoveJ home,v1000,z100,Pinza_2_1\WObj:=Workobject_2;
  ENDPROC
  PROC c_10()
    MoveJ home,v1000,z100,Pinza_2_1\WObj:=Workobject_2;
    MoveL c10_a,v1000,z100,Pinza_2_1\WObj:=Workobject_2;
    MoveL c10,v1000,fine,Pinza_2_1\WObj:=Workobject_2;
    MoveL c10_a,v1000,z100,Pinza_2_1\WObj:=Workobject_2;
    MoveJ home,v1000,z100,Pinza_2_1\WObj:=Workobject_2;
  ENDPROC
  PROC torno()
    MoveJ home_2,v1000,z100,Pinza_1\WObj:=Workobject_4;
    MoveJ prehome,v1000,z100,Pinza_1\WObj:=Workobject_4;
    MoveL fin_a,v1000,z100,Pinza_1\WObj:=Workobject_4;
    MoveL fin,v1000,fine,Pinza_1\WObj:=Workobject_4;
    WaitTime 1;
    MoveL fin_a,v1000,z100,Pinza_1\WObj:=Workobject_4;
  ENDPROC
  PROC giro()
    MoveJ final_a,v1000,z100,Pinza_2_1\WObj:=Workobject_2;
    MoveL final,v1000,fine,Pinza_2_1\WObj:=Workobject_2;
    WaitTime 1;
    MoveL final_a,v1000,z100,Pinza_2_1\WObj:=Workobject_2;
    MoveL home,v1000,z100,Pinza_2_1\WObj:=Workobject_2;
  ENDPROC
  PROC Path_10()
    MoveJ final_a,v1000,z100,tool0\WObj:=Workobject_2;
    MoveJ final,v1000,z100,tool0\WObj:=Workobject_2;
    MoveJ final_a,v1000,z100,tool0\WObj:=Workobject_2;
    MoveJ home,v1000,z100,tool0\WObj:=Workobject_2;
  ENDPROC
  PROC c_1_2()
    MoveJ home_2,v1000,z100,Pinza_1\WObj:=Workobject_4;
    MoveL c1a_3,v1000,fine,Pinza_1\WObj:=Workobject_4;
    MoveL c1_3,v1000,fine,Pinza_1\WObj:=Workobject_4;
    MoveL c1a_3,v1000,fine,Pinza_1\WObj:=Workobject_4;
    MoveL home_2,v1000,fine,Pinza_1\WObj:=Workobject_4;
  ENDPROC
  PROC c_2_2()
    MoveJ home_2,v1000,z100,Pinza_1\WObj:=Workobject_4;
    MoveL c2_a_2,v1000,fine,Pinza_1\WObj:=Workobject_4;
    MoveL c2_3,v1000,fine,Pinza_1\WObj:=Workobject_4;
    MoveL c2_a_2,v1000,fine,Pinza_1\WObj:=Workobject_4;
    MoveL home_2,v1000,fine,Pinza_1\WObj:=Workobject_4;
  ENDPROC
  PROC c_3_2()
    MoveJ sing,v1000,z100,Pinza_1\WObj:=Workobject_4;
    MoveJ c3_a_2_2,v1000,z100,Pinza_1\WObj:=Workobject_4;
    MoveJ c3_a_2,v1000,z100,Pinza_1\WObj:=Workobject_4;
    MoveL c3_3,v1000,fine,Pinza_1\WObj:=Workobject_4;
    MoveJ c3_a_2,v1000,z100,Pinza_1\WObj:=Workobject_4;
    MoveJ c3_a_2_2,v1000,z100,Pinza_1\WObj:=Workobject_4;
    MoveJ home_2,v1000,z100,Pinza_1\WObj:=Workobject_4;
  ENDPROC
  PROC c_4_2()
    MoveJ home_2,v1000,z100,Pinza_1\WObj:=Workobject_4;
    MoveL c4_a_2,v1000,fine,Pinza_1\WObj:=Workobject_4;
    MoveL c4_3,v1000,fine,Pinza_1\WObj:=Workobject_4;
    MoveL c4_a_2,v1000,fine,Pinza_1\WObj:=Workobject_4;
    MoveL home_2,v1000,fine,Pinza_1\WObj:=Workobject_4;
  ENDPROC
  PROC c_5_2()
    MoveJ home_2,v1000,z100,Pinza_1\WObj:=Workobject_4;
    MoveL c5_a_2,v1000,fine,Pinza_1\WObj:=Workobject_4;
    MoveL c5_3,v1000,fine,Pinza_1\WObj:=Workobject_4;
    MoveL c5_a_2,v1000,fine,Pinza_1\WObj:=Workobject_4;
    MoveL home_2,v1000,fine,Pinza_1\WObj:=Workobject_4;
  ENDPROC
  PROC c_6_2()
    MoveJ home_2,v1000,z100,Pinza_1\WObj:=Workobject_4;
    MoveL c6_a_2,v1000,fine,Pinza_1\WObj:=Workobject_4;
    MoveL c6_3,v1000,fine,Pinza_1\WObj:=Workobject_4;
    MoveL c6_a_2,v1000,fine,Pinza_1\WObj:=Workobject_4;
    MoveL home_2,v1000,fine,Pinza_1\WObj:=Workobject_4;
  ENDPROC
  PROC c_7_2()
    MoveJ home_2,v1000,z100,Pinza_1\WObj:=Workobject_4;
    MoveL c7_a_2,v1000,fine,Pinza_1\WObj:=Workobject_4;
    MoveL c7_3,v1000,fine,Pinza_1\WObj:=Workobject_4;
    MoveL c7_a_2,v1000,fine,Pinza_1\WObj:=Workobject_4;
    MoveL home_2,v1000,fine,Pinza_1\WObj:=Workobject_4;
  ENDPROC
  PROC c_8_2()
    MoveJ home_2,v1000,z100,Pinza_1\WObj:=Workobject_4;
    MoveJ sing_8,v1000,z100,Pinza_1\WObj:=Workobject_4;
    MoveJ c8_a_2,v1000,z100,Pinza_1\WObj:=Workobject_4;
    MoveL c8_3,v1000,fine,Pinza_1\WObj:=Workobject_4;
    MoveJ c8_a_2,v1000,z100,Pinza_1\WObj:=Workobject_4;
    MoveJ sing_8,v1000,z100,Pinza_1\WObj:=Workobject_4;
    MoveJ home_2,v1000,z100,Pinza_1\WObj:=Workobject_4;
  ENDPROC
  PROC c_9_2()
    MoveJ home_2,v1000,z100,Pinza_1\WObj:=Workobject_4;
    MoveL c9_a_3,v1000,fine,Pinza_1\WObj:=Workobject_4;
    MoveL c9_2,v1000,fine,Pinza_1\WObj:=Workobject_4;
    MoveL c9_a_3,v1000,fine,Pinza_1\WObj:=Workobject_4;
    MoveL home_2,v1000,fine,Pinza_1\WObj:=Workobject_4;
  ENDPROC
  PROC c_10_2()
    MoveJ home_2,v1000,z100,Pinza_1\WObj:=Workobject_4;
    MoveJ c10_a_2,v1000,z100,Pinza_1\WObj:=Workobject_4;
    MoveL c10_3,v1000,fine,Pinza_1\WObj:=Workobject_4;
    MoveJ c10_a_2,v1000,z100,Pinza_1\WObj:=Workobject_4;
    MoveL home_2,v1000,fine,Pinza_1\WObj:=Workobject_4;
  ENDPROC
  PROC limpieza()
    MoveL Target_20,v1000,fine,Soplador\WObj:=Workobject_5;
    MoveL Target_10,v1000,fine,Soplador\WObj:=Workobject_5;
    MoveL Target_10_2,v1000,fine,Soplador\WObj:=Workobject_5;
    MoveC Target_10_3,Target_10,v1000,fine,Soplador\WObj:=Workobject_5;
    MoveL Target_20,v1000,fine,Soplador\WObj:=Workobject_5;
  ENDPROC
  PROC main()
    c_1;
    torno;
    limpieza;
    giro;
    c_1_2;
    c_2;
    torno;
    limpieza;
    giro;
    c_2_2;
    c_3;
    torno;
    limpieza;
    giro;
    c_3_2;
    c_4;
    torno;
    limpieza;
    giro;
    c_4_2;
    c_5;
    torno;
    limpieza;
    giro;
    c_5_2;
    c_6;
    torno;
    limpieza;
    giro;
    c_6_2;
    c_7;
    torno;
    limpieza;
    giro;
    c_7_2;
    c_8;
    torno;
    limpieza;
    giro;
    c_8_2;
    c_9;
    torno;
    limpieza;
    giro;
    c_9_2;
    c_10;
    torno;
    limpieza;
    giro;
    c_10_2;
  ENDPROC
  PROC giro_mesa90()
    MoveL Target_30_3,v1000,fine,Vara\WObj:=Workobject_6;
    MoveL Target_30_2,v1000,fine,Vara\WObj:=Workobject_6;
    MoveC Target_50,Target_40_2,v1000,fine,Vara\WObj:=Workobject_6;
    MoveL Target_40_3,v1000,fine,Vara\WObj:=Workobject_6;
  ENDPROC
  PROC giro_mesa180()
    MoveL Target_60_2,v1000,fine,Vara\WObj:=Workobject_6;
    MoveL Target_60,v1000,fine,Vara\WObj:=Workobject_6;
    MoveL Target_60_3,v1000,fine,Vara\WObj:=Workobject_6;
    MoveL Target_30_3,v1000,fine,Vara\WObj:=Workobject_6;
    MoveL Target_30_2,v1000,fine,Vara\WObj:=Workobject_6;
    MoveC Target_50,Target_40_2,v1000,fine,Vara\WObj:=Workobject_6;
    MoveL Target_40_3,v1000,fine,Vara\WObj:=Workobject_6;
  ENDPROC
ENDMODULE

! task T_ROB1
MODULE CalibData
  TASK PERS wobjdata Workobject_2:=[FALSE,TRUE,"",[[0,0,0],[1,0,0,0]],[[0,0,0],[1,0,0,0]]];
  TASK PERS wobjdata Workobject_4:=[FALSE,TRUE,"",[[0,0,0],[1,0,0,0]],[[0,0,0],[1,0,0,0]]];
  PERS tooldata Pinza_2_1:=[TRUE,[[140,0,70],[0.707107,0,0.707107,0]],[1,[0,0,1],[1,0,0,0],0,0,0]];
  PERS tooldata Pinza_1:=[TRUE,[[-100,0,70],[0.707107,0,-0.707107,0]],[1,[0,0,1],[1,0,0,0],0,0,0]];
  PERS tooldata Vara:=[TRUE,[[0,0,250],[0.707107,0,0,0.707107]],[1,[0,0,1],[1,0,0,0],0,0,0]];
  PERS tooldata Soplador:=[TRUE,[[0,-70,70],[0.5,0.5,-0.5,0.5]],[1,[0,0,1],[1,0,0,0],0,0,0]];
  TASK PERS wobjdata Workobject_5:=[FALSE,TRUE,"",[[0,0,0],[1,0,0,0]],[[0,0,0],[1,0,0,0]]];
  TASK PERS wobjdata Workobject_6:=[FALSE,TRUE,"",[[0,0,0],[1,0,0,0]],[[0,0,0],[1,0,0,0]]];
ENDMODULE

